(* IEC 61131-3 sources: CodesysTest/alpha/export/FBs/Components/Indication/FB_K50_Button/Basic Mode, 1 file *)

(* ---- FB_K50_Button_BasicMode.pou.st ---- *)
(*#-#-#-#-#-#-#-#-#-#---Declaration---#-#-#-#-#-#-#-#-#-#-#-#-#*)

FUNCTION_BLOCK FB_K50_Button_BasicMode
VAR_INPUT
	baggerReady : BOOL;
	baggerFaulted : BOOL;
	baggerInCycle : BOOL;
END_VAR
VAR_OUTPUT
	IOLinkStateOutput : BYTE;
END_VAR
VAR
END_VAR
(*#-#-#-#-#-#-#-#-#-#---Implementation---#-#-#-#-#-#-#-#-#-#-#-#-#*)

IOLinkStateOutput := 0;
IF baggerReady THEN
	IOLinkStateOutput := 1;
END_IF
IF baggerInCycle THEN
	IOLinkStateOutput := 2;
END_IF
IF baggerFaulted THEN
	IOLinkStateOutput := 3;
END_IF
